(* IEC 61131-3 sources: AXOpen/src/components.abstractions/ctrl/src/AxoDrives (part 4) *)

        ///<summary>
        /// This method presents general axis errors not relating to the methods.
        /// (for instance axis errors, drive errors, communication errors)
        /// This vendor specific method must be overridden in the derived class.
        ///<summary>
        METHOD PUBLIC ABSTRACT MC_ReadAxisError
            VAR_IN_OUT
                AxisRef         :   AxoAxisRef;                 //  Reference to the axis
            END_VAR
            VAR_INPUT
                Enable          :   BOOL;                       //  Get the value of the parameter continuously while enabled
            END_VAR
            VAR_OUTPUT
                Valid           :   BOOL;                       //  A valid output is available at the method
                Busy            :   BOOL;                       //  The method is not finished and new output values are to be expected
                Error           :   BOOL;                       //  Signals that an error has occurred within the method
                ErrorID         :   WORD;                       //  Error identification
                AxisErrorID     :   WORD;                       //  The value of the axis error. These values are vendor specific
            END_VAR
        END_METHOD

        ///<summary>
        /// This method makes the transition from the state ‘ErrorStop’ to ‘Standstill’ or ‘Disabled’ by resetting all
        /// internal axis-related errors – it does not affect the output of the other methods.
        /// This vendor specific method must be overridden in the derived class.
        ///<summary>
        METHOD PUBLIC ABSTRACT MC_Reset
            VAR_IN_OUT
                AxisRef         :   AxoAxisRef;                 //  Reference to the axis
            END_VAR
            VAR_INPUT
                Execute         :   BOOL;                       //  Resets all internal axis-related error
            END_VAR
            VAR_OUTPUT
                Done            :   BOOL;                       //  ‘Standstill’ or ‘Disabled’ state is reached
                Busy            :   BOOL;                       //  The method is not finished and new output values are to be expected
                Error           :   BOOL;                       //  Signals that an error has occurred within the method
                ErrorID         :   WORD;                       //  Error identification
            END_VAR
        END_METHOD
    END_CLASS
END_NAMESPACE

(* ---- AxoDrive_Config.st ---- *)
NAMESPACE AXOpen.Components.Abstractions.AxoDrives
    {#ix-attr:[Container(Layout.Wrap)]}
    CLASS AxoDrive_Config
        VAR PUBLIC
            {#ix-set:AttributeName = "<#Info time#>"}
            InfoTime : LTIME := LT#2S;
            {#ix-set:AttributeName = "<#Error time#>"}
            ErrorTime : LTIME := LT#5S;
        END_VAR
    END_CLASS
END_NAMESPACE

(* ---- AxoDrive_Status.st ---- *)
USING AXOpen.Core;
NAMESPACE AXOpen.Components.Abstractions.AxoDrives
    {#ix-attr:[Container(Layout.Stack)]}
    CLASS AxoDrive_Status EXTENDS AXOpen.Components.Abstractions.AxoComponent_Status
        VAR PUBLIC
            {#ix-attr:[ReadOnly()]}
            CurrentMotionTaskId    :   INT;
        END_VAR
    END_CLASS
END_NAMESPACE

(* ---- AxoDriveParameterChannelIDN.st ---- *)
USING AXOpen.Core;
NAMESPACE AXOpen.Components.Abstractions.AxoDrives
    CLASS AxoDriveParameterChannelIdnIn
        VAR PUBLIC
            StatusWord  :   WORD;
            Index       :   WORD;
            SubIndex    :   WORD;
            ValueHigh   :   WORD;
            ValueLow    :   WORD;
        END_VAR
    END_CLASS
    CLASS AxoDriveParameterChannelIdnOut
        VAR PUBLIC
            ControlWord :   WORD;
            Index       :   WORD;
            SubIndex    :   WORD;
            ValueHigh   :   WORD;
            ValueLow    :   WORD;
        END_VAR
    END_CLASS
END_NAMESPACE

(* ---- AxoMotionExecutionTask.st ---- *)
USING AXOpen.Core;
USING AXOpen.Messaging;
USING AXOpen.Messaging.Static;

NAMESPACE AXOpen.Components.Abstractions.AxoDrives
    CLASS PUBLIC ABSTRACT AxoMotionExecutionTask EXTENDS AXOpen.Core.AxoTask
        VAR PUBLIC
            Messenger   :   AxoMessenger;
        END_VAR

        VAR PROTECTED
            _infoTimer      :   AXOpen.Timers.OnDelayTimer;
            _errorTimer     :   AXOpen.Timers.OnDelayTimer;
            _infoTime       :   LTIME := LT#2S;
            _errorTime      :   LTIME := LT#5S;
            _progress       :   INT;
        END_VAR
        VAR PRIVATE
            _motionTaskId   :   INT;
            _isBusyPV       :   BOOL;
        END_VAR

        ///<summary>
        /// Runs the logic of this tasks.
        /// >[!IMPORTANT] This method must be called cyclically.
        ///</summary>
        METHOD PUBLIC Run
            VAR_IN_OUT
                AxisRef :   AxoAxisRef;
            END_VAR

            VAR_OUTPUT
                Done            :   BOOL;   //Motion task syccesfully finished
                Busy            :   BOOL;   //The FB is not finished and new output values are to be expected
                Active          :   BOOL;   //Indicates that the FB has control on the axis
                CommandAborted  :   BOOL;   //‘Command’ is aborted by another command
                Error           :   BOOL;   //Signals that an error has occurred within the Function Block
                ErrorID         :   WORD;   //Error identification
            END_VAR

            VAR
                _Active         :   BOOL;
                _ErrorID        :   WORD;
            END_VAR

            _infoTime := AxisRef.Config.InfoTime;
            _errorTime := AxisRef.Config.ErrorTime;
            Messenger.Serve(THIS);
            _Active := FALSE;
            _ErrorID := WORD#0;

            // //Set the _motionTaskId for discovering which method controls the axis
            // IF _motionTaskId = 0 THEN
            //     AxisRef.Status._MotionTaskIds := AxisRef.Status._MotionTaskIds + 1;
            //     _motionTaskId  := AxisRef.Status._MotionTaskIds;
            // END_IF;

            _isBusyPV := THIS.IsBusy();
            IF THIS.Execute() THEN
                THIS.MotionTaskExecute(AxisRef,_Active,_ErrorID);
                THIS.CallTimers(TRUE);
            END_IF;

            THIS.MotionTaskCyclic(AxisRef,_Active,_ErrorID);

            //Set the _motionTaskId as current one at the begining of the motion task
            IF NOT _isBusyPV AND THIS.IsBusy() THEN
                AxisRef.Status._CurrentMotionTaskId := _motionTaskId;
            END_IF;

            Done            := THIS.IsDone();
            Busy            := THIS.IsBusy();
            Active          := _Active;
            CommandAborted  := THIS.IsAborted();
            Error           := THIS.HasError();
            ErrorID         := _ErrorID;
        END_METHOD

        METHOD PUBLIC ABSTRACT MotionTaskExecute
            VAR_IN_OUT
                AxisRef     :   AxoAxisRef;
                Active      :   BOOL;       //Indicates that the FB has control on the axis
                ErrorID     :   WORD;       //Error identification
            END_VAR
        END_METHOD

        METHOD PUBLIC ABSTRACT MotionTaskCyclic
            VAR_IN_OUT
                AxisRef     :   AxoAxisRef;
                Active      :   BOOL;       //Indicates that the FB has control on the axis
                ErrorID     :   WORD;       //Error identification
            END_VAR
        END_METHOD

        METHOD INTERNAL CallTimers
            VAR_INPUT
                signal : BOOL;
            END_VAR

            _infoTimer.OnDelay(THIS, signal , _infoTime);
            _errorTimer.OnDelay(THIS, signal , _errorTime );
        END_METHOD

        METHOD PUBLIC Restore
            _progress := 0;
            THIS.CallTimers(FALSE);
            SUPER.Restore();
        END_METHOD

        METHOD PROTECTED OVERRIDE OnRestore
            ;
        END_METHOD

        METHOD PROTECTED OVERRIDE OnAbort
            ;
        END_METHOD

        METHOD PROTECTED OVERRIDE OnDone
            ;
        END_METHOD

        METHOD PROTECTED OVERRIDE OnError
            ;
        END_METHOD

        METHOD PROTECTED OVERRIDE OnStart
            ;
        END_METHOD
    END_CLASS
END_NAMESPACE

(* ---- AxoMotionJogTask.st ---- *)
USING AXOpen.Core;

NAMESPACE AXOpen.Components.Abstractions.AxoDrives
    CLASS PUBLIC AxoMotionJogTask EXTENDS AXOpen.Core.AxoMomentaryTask
        VAR PUBLIC
            StartMotion :   BOOL;
            StopMotion  :   BOOL;
        END_VAR
        METHOD PROTECTED OVERRIDE OnSwitchedOn
            StartMotion :=  TRUE;
            StopMotion  :=  FALSE;
        END_METHOD
        METHOD PROTECTED OVERRIDE OnSwitchedOff
            StartMotion :=  FALSE;
            StopMotion  :=  TRUE;
        END_METHOD
    END_CLASS
END_NAMESPACE

(* ---- AxoMotionLevelTask.st ---- *)
USING AXOpen.Core;
USING AXOpen.Messaging;
USING AXOpen.Messaging.Static;

NAMESPACE AXOpen.Components.Abstractions.AxoDrives
    CLASS PUBLIC ABSTRACT AxoMotionLevelTask EXTENDS  AXOpen.Components.Abstractions.AxoDrives.AxoMotionStateTask
        ///<summary>
        /// Runs the logic of this tasks.
        /// >[!IMPORTANT] This method must be called cyclically.
        ///</summary>
        METHOD PUBLIC Run
            VAR_IN_OUT
                AxisRef :   AxoAxisRef;
            END_VAR
            VAR_INPUT
                Enable  : BOOL;
            END_VAR

            VAR_OUTPUT
                Busy            :   BOOL;   //  The FB is not finished and new output values are to be expected
                Valid           :   BOOL;   //  Valid set of outputs is available at the FB.
                Error           :   BOOL;   //  Signals that an error has occurred within the Function Block
                ErrorID         :   WORD;   //  Error identification
            END_VAR

            SUPER.Run(AxisRef,Busy,Valid,Error,ErrorID);

            IF Enable THEN
                SUPER.SwitchOn();
            ELSE
                SUPER.SwitchOff();
            END_IF;

            THIS.Cyclic();

        END_METHOD

        METHOD PUBLIC ABSTRACT Cyclic
        END_METHOD

    END_CLASS
END_NAMESPACE

(* ---- AxoMotionStateTask.st ---- *)
USING AXOpen.Core;
USING AXOpen.Messaging;
USING AXOpen.Messaging.Static;

NAMESPACE AXOpen.Components.Abstractions.AxoDrives
    CLASS PUBLIC ABSTRACT AxoMotionStateTask EXTENDS AXOpen.Core.AxoToggleTask
        VAR PUBLIC
            Messenger   :   AxoMessenger;
        END_VAR

        ///<summary>
        /// Runs the logic of this tasks.
        /// >[!IMPORTANT] This method must be called cyclically.
        ///</summary>
        METHOD PUBLIC Run
            VAR_IN_OUT
                AxisRef :   AxoAxisRef;
            END_VAR

            VAR_OUTPUT
                Busy            :   BOOL;   //  The FB is not finished and new output values are to be expected
                Valid           :   BOOL;   //  Valid set of outputs is available at the FB.
                Error           :   BOOL;   //  Signals that an error has occurred within the Function Block
                ErrorID         :   WORD;   //  Error identification
            END_VAR

            VAR
                _Busy           :   BOOL;
                _Valid          :   BOOL;
                _Error          :   BOOL;
                _ErrorID        :   WORD;
            END_VAR

            Messenger.Serve(THIS);
            _Busy := FALSE;
            _Valid := FALSE;
            _Error := FALSE;
            _ErrorID := WORD#0;

            IF THIS.IsSwitchedOn() THEN
                THIS.StateTaskOn(AxisRef,_Busy,_Valid,_Error,_ErrorID);
            ELSE
                THIS.StateTaskOff(AxisRef,_Busy,_Valid,_Error,_ErrorID);
            END_IF;

            Busy        := _Busy;
            Valid       := _Valid;
            Error       := _Error;
            ErrorID     := _ErrorID;
        END_METHOD

        METHOD PUBLIC ABSTRACT StateTaskOn
            VAR_IN_OUT
                AxisRef     :   AxoAxisRef;
                Busy        :   BOOL;   //  The FB is not finished and new output values are to be expected
                Valid       :   BOOL;   //  Valid set of outputs is available at the FB.
                Error       :   BOOL;   //  Signals that an error has occurred within the Function Block
                ErrorID     :   WORD;   //  Error identification
            END_VAR
        END_METHOD

        METHOD PUBLIC ABSTRACT StateTaskOff
            VAR_IN_OUT
                AxisRef     :   AxoAxisRef;
                Busy        :   BOOL;   //  The FB is not finished and new output values are to be expected
                Valid       :   BOOL;   //  Valid set of outputs is available at the FB.
                Error       :   BOOL;   //  Signals that an error has occurred within the Function Block
                ErrorID     :   WORD;   //  Error identification
            END_VAR
        END_METHOD
    END_CLASS
END_NAMESPACE

(* ---- AxoPower.st ---- *)
USING AXOpen.Core;
USING AXOpen.Messaging;
USING AXOpen.Messaging.Static;

NAMESPACE AXOpen.Components.Abstractions.AxoDrives
    CLASS PUBLIC AxoPower EXTENDS AXOpen.Core.AxoToggleTask
        VAR PRIVATE
            _motionTaskId    :  AXOpen.Components.Abstractions.AxoDrives.eAxoMotionTaskId := AXOpen.Components.Abstractions.AxoDrives.eAxoMotionTaskId#Axo_Power;
            _EnablePositive  :  AXOpen.Core.AxoToggleTask;
            _EnableNegative  :  AXOpen.Core.AxoToggleTask;
            _manualOverride  :  BOOL;
        END_VAR

        ///<summary>
        /// Runs the logic of this tasks.
        /// >[!IMPORTANT] This method must be called cyclically.
        ///</summary>
        METHOD PUBLIC Run
            // VAR_IN_OUT
            //     AxisRef :   AxoAxisRef;
            // END_VAR
            VAR_INPUT
                Enable          :   BOOL;                       //  As long as ‘Enable’ is true, power is being enabled.
                EnablePositive  :   BOOL;                       //  As long as ‘Enable’ is true, this permits motion in positive direction
                EnableNegative  :   BOOL;                       //  As long as ‘Enable’ is true, this permits motion in negative direction
            END_VAR

            SUPER.Run();

            // Enables manually switch off and switch on the power in case of enable is 'TRUE'
            IF _manualOverride THEN
                SUPER.SetIsDisabled(NOT Enable);
            ELSE
                SUPER.SetIsDisabled(FALSE);
                IF Enable THEN
                    SUPER.SwitchOn();
                ELSE
                    SUPER.SwitchOff();
                END_IF;
            END_IF;

            _EnablePositive.Initialize(THIS);
            _EnablePositive.Run();
            _EnablePositive.SetIsDisabled(SUPER.IsSwitchedOn());
            IF EnablePositive THEN
                _EnablePositive.SwitchOn();
            ELSE
                _EnablePositive.SwitchOff();
            END_IF;

            _EnableNegative.Initialize(THIS);
            _EnableNegative.Run();
            _EnableNegative.SetIsDisabled(SUPER.IsSwitchedOn());
            IF EnableNegative THEN
                _EnableNegative.SwitchOn();
            ELSE
                _EnableNegative.SwitchOff();
            END_IF;

            _manualOverride := FALSE;
        END_METHOD

        ///<summary>
        /// Returns `TRUE` if movement to positive direction is enabled
        ///</summary>
        METHOD PUBLIC EnabledPositive : BOOL
            EnabledPositive := _EnablePositive.IsSwitchedOn();
        END_METHOD
        ///<summary>
        /// Returns `TRUE` if movement to positive direction is disabled
        ///</summary>
        METHOD PUBLIC DisabledPositive : BOOL
            DisabledPositive := _EnablePositive.IsSwitchedOff();
        END_METHOD
        ///<summary>
        /// Returns `TRUE` if movement to negative direction is enabled
        ///</summary>
        METHOD PUBLIC EnabledNegative : BOOL
            EnabledNegative := _EnableNegative.IsSwitchedOn();
        END_METHOD
        ///<summary>
        /// Returns `TRUE` if movement to negative direction is disabled
        ///</summary>
        METHOD PUBLIC DisabledNegative : BOOL
            DisabledNegative := _EnableNegative.IsSwitchedOff();
        END_METHOD

        METHOD PUBLIC Manual
            _manualOverride := TRUE;
        END_METHOD
    END_CLASS
END_NAMESPACE
